// TIA Portal V17 export
// export: Created 2023-05-12T10:40:25.6107869Z, DisplayName Totally Integrated Automation Portal, DisplayVersion V17 Update 4, DisplayName TIA Portal Openness, DisplayVersion V17 Update 4, DisplayName TIA Portal Version Control Interface, DisplayVersion V17, DisplayName STEP 7 Professional, DisplayVersion V17 Update 4, DisplayName STEP 7 Safety, DisplayVersion V17, DisplayName WinCC Advanced / Unified PC, DisplayVersion V17 Update 4
FUNCTION_BLOCK "FB_EM_InputConditioning"   // FB19, LAD
{ S7_Optimized_Access := 'TRUE' }
VERSION : 0.1
// stored: AutoNumber true, CodeModifiedDate 2023-05-12T12:59:41.6492354Z, CompileDate 2023-05-12T12:59:41.6492354Z, CreationDate 2023-05-08T12:19:11.3376827Z, DownloadWithoutReinit false, HandleErrorsWithinBlock false, InterfaceModifiedDate 2023-05-12T12:59:19.7337351Z, IsConsistent true, IsIECCheckEnabled false, IsKnowHowProtected false, IsRetainMemResEnabled false, IsWriteProtected false, LibraryConformanceStatus Warning: The object contains access to global data blocks., MemoryReserve 100, ModifiedDate 2023-05-12T12:59:41.6492354Z, ParameterModified 2022-09-13T10:25:33.4387708Z, PLCSimAdvancedSupport true, SetENOAutomatically false, StructureModified 2023-05-12T12:59:19.7337351Z, UDAEnableTagReadback false
   VAR
      TT01_TempZasil_JKK13_Inst { S7_SetPoint := 'True'} : "FB_CM_MeasurementPoint";
      TT02_TempPowr_JKK13_Inst { S7_SetPoint := 'True'} : "FB_CM_MeasurementPoint";
      TT03_TemZasil_SPC_Kart_Inst { S7_SetPoint := 'True'} : "FB_CM_MeasurementPoint";
      TT04_TempPowr_SPC_Kart_Inst { S7_SetPoint := 'True'} : "FB_CM_MeasurementPoint";
      TT05_TempZasil_SC_Rogacz_Inst { S7_SetPoint := 'True'} : "FB_CM_MeasurementPoint";
      TT06_TempPowr_SC_Rogacz_Inst { S7_SetPoint := 'True'} : "FB_CM_MeasurementPoint";
      PT01_CisnZasil_JKK13_Inst { S7_SetPoint := 'True'} : "FB_CM_MeasurementPoint";
      PT02_CisnPowr_JKK13_Inst { S7_SetPoint := 'True'} : "FB_CM_MeasurementPoint";
      PT03_CisnZasil_SPC_Kart_Inst { S7_SetPoint := 'True'} : "FB_CM_MeasurementPoint";
      PT04_CisnPowr_SPC_Kart_Inst { S7_SetPoint := 'True'} : "FB_CM_MeasurementPoint";
      PT05_CisnZasil_SC_Rogacz_Inst { S7_SetPoint := 'True'} : "FB_CM_MeasurementPoint";
      PT06_CisnPowr_SC_Rogacz_Inst { S7_SetPoint := 'True'} : "FB_CM_MeasurementPoint";
      TTs_TempSzafy_Inst { S7_SetPoint := 'True'} : "FB_CM_MeasurementPoint";
      TTk_TempKom_Inst { S7_SetPoint := 'True'} : "FB_CM_MeasurementPoint";
      TTz_TempZewn_Inst { S7_SetPoint := 'True'} : "FB_CM_MeasurementPoint";
      Rezerwa1_Inst { S7_SetPoint := 'True'} : "FB_CM_MeasurementPoint";
   END_VAR
BEGIN

REGION Network 1: TT01_TempZasil_JKK13 - Temperatura zasilania z JKK13
   // TT01_TempZasil_JKK13 - Temperatura zasilania z JKK13
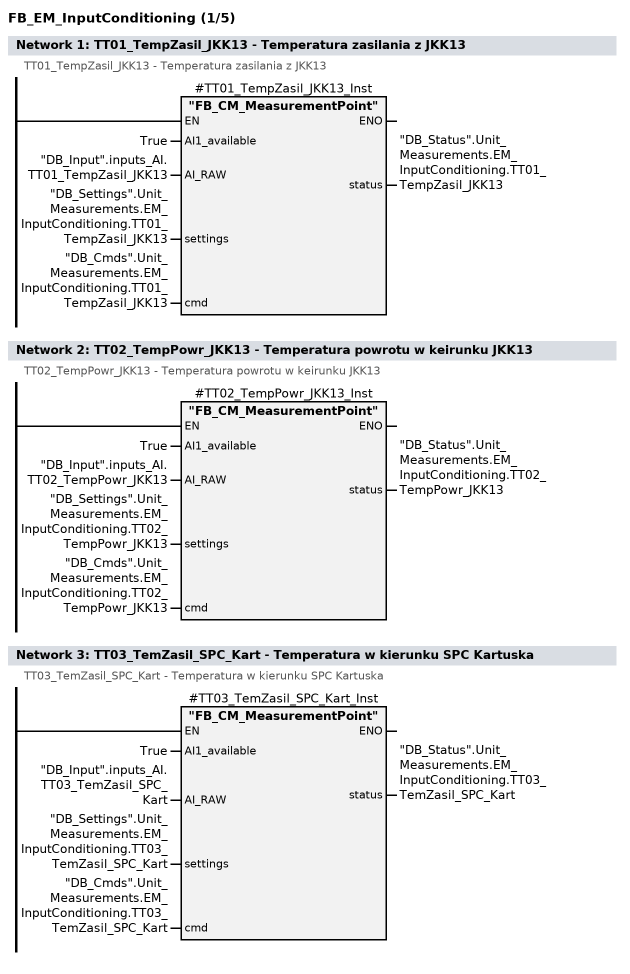
   RUNG wire#powerrail
      #TT01_TempZasil_JKK13_Inst(AI1_available := True, AI_RAW := "DB_Input".inputs_AI.TT01_TempZasil_JKK13, settings := "DB_Settings".Unit_Measurements.EM_InputConditioning.TT01_TempZasil_JKK13, cmd := "DB_Cmds".Unit_Measurements.EM_InputConditioning.TT01_TempZasil_JKK13, status => "DB_Status".Unit_Measurements.EM_InputConditioning.TT01_TempZasil_JKK13)
   END_RUNG
   // the same network as SCL:
   #TT01_TempZasil_JKK13_Inst(AI1_available := True,   // "FB_CM_MeasurementPoint"
                           AI_RAW := "DB_Input".inputs_AI.TT01_TempZasil_JKK13,
                           settings := "DB_Settings".Unit_Measurements.EM_InputConditioning.TT01_TempZasil_JKK13,
                           cmd := "DB_Cmds".Unit_Measurements.EM_InputConditioning.TT01_TempZasil_JKK13,
                           status => "DB_Status".Unit_Measurements.EM_InputConditioning.TT01_TempZasil_JKK13);
END_REGION

REGION Network 2: TT02_TempPowr_JKK13 - Temperatura powrotu w keirunku JKK13
   // TT02_TempPowr_JKK13 - Temperatura powrotu w keirunku JKK13
   RUNG wire#powerrail
      #TT02_TempPowr_JKK13_Inst(AI1_available := True, AI_RAW := "DB_Input".inputs_AI.TT02_TempPowr_JKK13, settings := "DB_Settings".Unit_Measurements.EM_InputConditioning.TT02_TempPowr_JKK13, cmd := "DB_Cmds".Unit_Measurements.EM_InputConditioning.TT02_TempPowr_JKK13, status => "DB_Status".Unit_Measurements.EM_InputConditioning.TT02_TempPowr_JKK13)
   END_RUNG
   // the same network as SCL:
   #TT02_TempPowr_JKK13_Inst(AI1_available := True,   // "FB_CM_MeasurementPoint"
                           AI_RAW := "DB_Input".inputs_AI.TT02_TempPowr_JKK13,
                           settings := "DB_Settings".Unit_Measurements.EM_InputConditioning.TT02_TempPowr_JKK13,
                           cmd := "DB_Cmds".Unit_Measurements.EM_InputConditioning.TT02_TempPowr_JKK13,
                           status => "DB_Status".Unit_Measurements.EM_InputConditioning.TT02_TempPowr_JKK13);
END_REGION

REGION Network 3: TT03_TemZasil_SPC_Kart - Temperatura w kierunku SPC Kartuska
   // TT03_TemZasil_SPC_Kart - Temperatura w kierunku SPC Kartuska
   RUNG wire#powerrail
      #TT03_TemZasil_SPC_Kart_Inst(AI1_available := True, AI_RAW := "DB_Input".inputs_AI.TT03_TemZasil_SPC_Kart, settings := "DB_Settings".Unit_Measurements.EM_InputConditioning.TT03_TemZasil_SPC_Kart, cmd := "DB_Cmds".Unit_Measurements.EM_InputConditioning.TT03_TemZasil_SPC_Kart, status => "DB_Status".Unit_Measurements.EM_InputConditioning.TT03_TemZasil_SPC_Kart)
   END_RUNG
   // the same network as SCL:
   #TT03_TemZasil_SPC_Kart_Inst(AI1_available := True,   // "FB_CM_MeasurementPoint"
                           AI_RAW := "DB_Input".inputs_AI.TT03_TemZasil_SPC_Kart,
                           settings := "DB_Settings".Unit_Measurements.EM_InputConditioning.TT03_TemZasil_SPC_Kart,
                           cmd := "DB_Cmds".Unit_Measurements.EM_InputConditioning.TT03_TemZasil_SPC_Kart,
                           status => "DB_Status".Unit_Measurements.EM_InputConditioning.TT03_TemZasil_SPC_Kart);
END_REGION

REGION Network 4: TT04_TempPowr_SPC_Kart - Temperatura powrotu z SPC Kartuska
   // TT04_TempPowr_SPC_Kart - Temperatura powrotu z SPC Kartuska
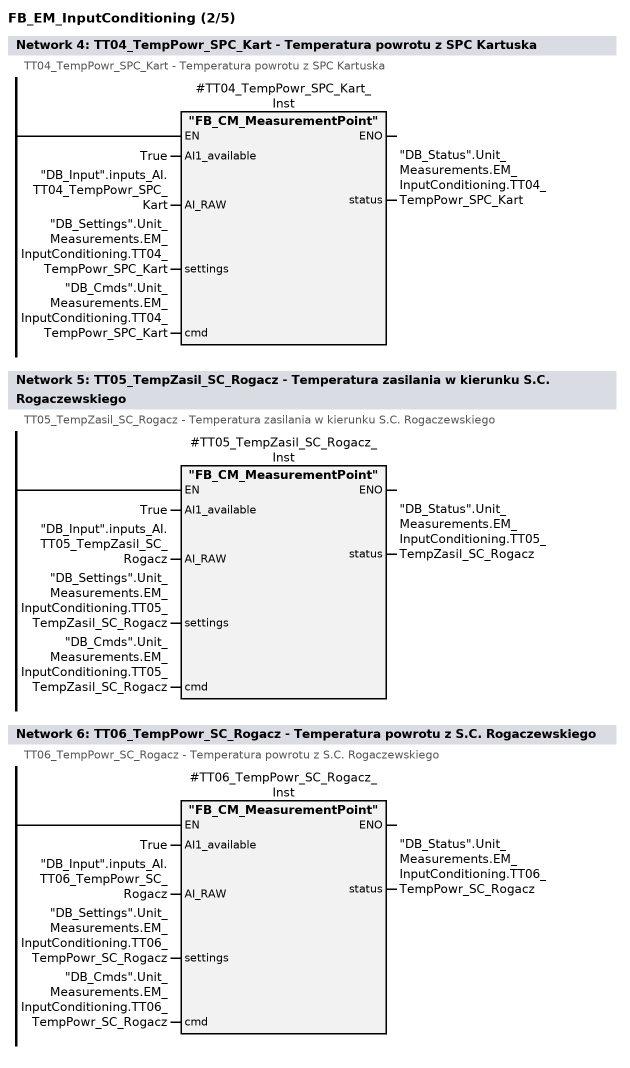
   RUNG wire#powerrail
      #TT04_TempPowr_SPC_Kart_Inst(AI1_available := True, AI_RAW := "DB_Input".inputs_AI.TT04_TempPowr_SPC_Kart, settings := "DB_Settings".Unit_Measurements.EM_InputConditioning.TT04_TempPowr_SPC_Kart, cmd := "DB_Cmds".Unit_Measurements.EM_InputConditioning.TT04_TempPowr_SPC_Kart, status => "DB_Status".Unit_Measurements.EM_InputConditioning.TT04_TempPowr_SPC_Kart)
   END_RUNG
   // the same network as SCL:
   #TT04_TempPowr_SPC_Kart_Inst(AI1_available := True,   // "FB_CM_MeasurementPoint"
                           AI_RAW := "DB_Input".inputs_AI.TT04_TempPowr_SPC_Kart,
                           settings := "DB_Settings".Unit_Measurements.EM_InputConditioning.TT04_TempPowr_SPC_Kart,
                           cmd := "DB_Cmds".Unit_Measurements.EM_InputConditioning.TT04_TempPowr_SPC_Kart,
                           status => "DB_Status".Unit_Measurements.EM_InputConditioning.TT04_TempPowr_SPC_Kart);
END_REGION

REGION Network 5: TT05_TempZasil_SC_Rogacz - Temperatura zasilania w kierunku S.C. Rogaczewskiego
   // TT05_TempZasil_SC_Rogacz - Temperatura zasilania w kierunku S.C. Rogaczewskiego
   RUNG wire#powerrail
      #TT05_TempZasil_SC_Rogacz_Inst(AI1_available := True, AI_RAW := "DB_Input".inputs_AI.TT05_TempZasil_SC_Rogacz, settings := "DB_Settings".Unit_Measurements.EM_InputConditioning.TT05_TempZasil_SC_Rogacz, cmd := "DB_Cmds".Unit_Measurements.EM_InputConditioning.TT05_TempZasil_SC_Rogacz, status => "DB_Status".Unit_Measurements.EM_InputConditioning.TT05_TempZasil_SC_Rogacz)
   END_RUNG
   // the same network as SCL:
   #TT05_TempZasil_SC_Rogacz_Inst(AI1_available := True,   // "FB_CM_MeasurementPoint"
                           AI_RAW := "DB_Input".inputs_AI.TT05_TempZasil_SC_Rogacz,
                           settings := "DB_Settings".Unit_Measurements.EM_InputConditioning.TT05_TempZasil_SC_Rogacz,
                           cmd := "DB_Cmds".Unit_Measurements.EM_InputConditioning.TT05_TempZasil_SC_Rogacz,
                           status => "DB_Status".Unit_Measurements.EM_InputConditioning.TT05_TempZasil_SC_Rogacz);
END_REGION

REGION Network 6: TT06_TempPowr_SC_Rogacz - Temperatura powrotu z S.C. Rogaczewskiego
   // TT06_TempPowr_SC_Rogacz - Temperatura powrotu z S.C. Rogaczewskiego
   RUNG wire#powerrail
      #TT06_TempPowr_SC_Rogacz_Inst(AI1_available := True, AI_RAW := "DB_Input".inputs_AI.TT06_TempPowr_SC_Rogacz, settings := "DB_Settings".Unit_Measurements.EM_InputConditioning.TT06_TempPowr_SC_Rogacz, cmd := "DB_Cmds".Unit_Measurements.EM_InputConditioning.TT06_TempPowr_SC_Rogacz, status => "DB_Status".Unit_Measurements.EM_InputConditioning.TT06_TempPowr_SC_Rogacz)
   END_RUNG
   // the same network as SCL:
   #TT06_TempPowr_SC_Rogacz_Inst(AI1_available := True,   // "FB_CM_MeasurementPoint"
                           AI_RAW := "DB_Input".inputs_AI.TT06_TempPowr_SC_Rogacz,
                           settings := "DB_Settings".Unit_Measurements.EM_InputConditioning.TT06_TempPowr_SC_Rogacz,
                           cmd := "DB_Cmds".Unit_Measurements.EM_InputConditioning.TT06_TempPowr_SC_Rogacz,
                           status => "DB_Status".Unit_Measurements.EM_InputConditioning.TT06_TempPowr_SC_Rogacz);
END_REGION

REGION Network 7: PT01_CisnZasil_JKK13 - CIśnienie zasilania z JKK13
   // PT01_CisnZasil_JKK13 - CIśnienie zasilania z JKK13
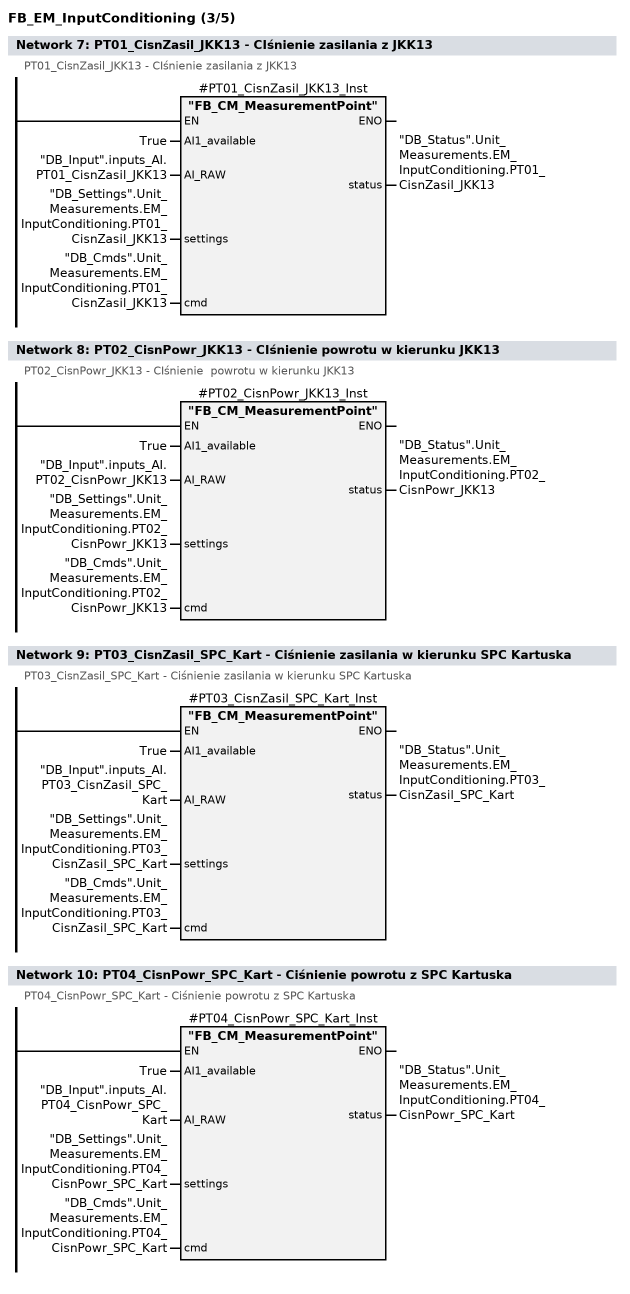
   RUNG wire#powerrail
      #PT01_CisnZasil_JKK13_Inst(AI1_available := True, AI_RAW := "DB_Input".inputs_AI.PT01_CisnZasil_JKK13, settings := "DB_Settings".Unit_Measurements.EM_InputConditioning.PT01_CisnZasil_JKK13, cmd := "DB_Cmds".Unit_Measurements.EM_InputConditioning.PT01_CisnZasil_JKK13, status => "DB_Status".Unit_Measurements.EM_InputConditioning.PT01_CisnZasil_JKK13)
   END_RUNG
   // the same network as SCL:
   #PT01_CisnZasil_JKK13_Inst(AI1_available := True,   // "FB_CM_MeasurementPoint"
                           AI_RAW := "DB_Input".inputs_AI.PT01_CisnZasil_JKK13,
                           settings := "DB_Settings".Unit_Measurements.EM_InputConditioning.PT01_CisnZasil_JKK13,
                           cmd := "DB_Cmds".Unit_Measurements.EM_InputConditioning.PT01_CisnZasil_JKK13,
                           status => "DB_Status".Unit_Measurements.EM_InputConditioning.PT01_CisnZasil_JKK13);
END_REGION

REGION Network 8: PT02_CisnPowr_JKK13 - CIśnienie powrotu w kierunku JKK13
   // PT02_CisnPowr_JKK13 - CIśnienie  powrotu w kierunku JKK13
   RUNG wire#powerrail
      #PT02_CisnPowr_JKK13_Inst(AI1_available := True, AI_RAW := "DB_Input".inputs_AI.PT02_CisnPowr_JKK13, settings := "DB_Settings".Unit_Measurements.EM_InputConditioning.PT02_CisnPowr_JKK13, cmd := "DB_Cmds".Unit_Measurements.EM_InputConditioning.PT02_CisnPowr_JKK13, status => "DB_Status".Unit_Measurements.EM_InputConditioning.PT02_CisnPowr_JKK13)
   END_RUNG
   // the same network as SCL:
   #PT02_CisnPowr_JKK13_Inst(AI1_available := True,   // "FB_CM_MeasurementPoint"
                           AI_RAW := "DB_Input".inputs_AI.PT02_CisnPowr_JKK13,
                           settings := "DB_Settings".Unit_Measurements.EM_InputConditioning.PT02_CisnPowr_JKK13,
                           cmd := "DB_Cmds".Unit_Measurements.EM_InputConditioning.PT02_CisnPowr_JKK13,
                           status => "DB_Status".Unit_Measurements.EM_InputConditioning.PT02_CisnPowr_JKK13);
END_REGION

REGION Network 9: PT03_CisnZasil_SPC_Kart - Ciśnienie zasilania w kierunku SPC Kartuska
   // PT03_CisnZasil_SPC_Kart - Ciśnienie zasilania w kierunku SPC Kartuska
   RUNG wire#powerrail
      #PT03_CisnZasil_SPC_Kart_Inst(AI1_available := True, AI_RAW := "DB_Input".inputs_AI.PT03_CisnZasil_SPC_Kart, settings := "DB_Settings".Unit_Measurements.EM_InputConditioning.PT03_CisnZasil_SPC_Kart, cmd := "DB_Cmds".Unit_Measurements.EM_InputConditioning.PT03_CisnZasil_SPC_Kart, status => "DB_Status".Unit_Measurements.EM_InputConditioning.PT03_CisnZasil_SPC_Kart)
   END_RUNG
   // the same network as SCL:
   #PT03_CisnZasil_SPC_Kart_Inst(AI1_available := True,   // "FB_CM_MeasurementPoint"
                           AI_RAW := "DB_Input".inputs_AI.PT03_CisnZasil_SPC_Kart,
                           settings := "DB_Settings".Unit_Measurements.EM_InputConditioning.PT03_CisnZasil_SPC_Kart,
                           cmd := "DB_Cmds".Unit_Measurements.EM_InputConditioning.PT03_CisnZasil_SPC_Kart,
                           status => "DB_Status".Unit_Measurements.EM_InputConditioning.PT03_CisnZasil_SPC_Kart);
END_REGION

REGION Network 10: PT04_CisnPowr_SPC_Kart - Ciśnienie powrotu z SPC Kartuska
   // PT04_CisnPowr_SPC_Kart - Ciśnienie powrotu z SPC Kartuska
   RUNG wire#powerrail
      #PT04_CisnPowr_SPC_Kart_Inst(AI1_available := True, AI_RAW := "DB_Input".inputs_AI.PT04_CisnPowr_SPC_Kart, settings := "DB_Settings".Unit_Measurements.EM_InputConditioning.PT04_CisnPowr_SPC_Kart, cmd := "DB_Cmds".Unit_Measurements.EM_InputConditioning.PT04_CisnPowr_SPC_Kart, status => "DB_Status".Unit_Measurements.EM_InputConditioning.PT04_CisnPowr_SPC_Kart)
   END_RUNG
   // the same network as SCL:
   #PT04_CisnPowr_SPC_Kart_Inst(AI1_available := True,   // "FB_CM_MeasurementPoint"
                           AI_RAW := "DB_Input".inputs_AI.PT04_CisnPowr_SPC_Kart,
                           settings := "DB_Settings".Unit_Measurements.EM_InputConditioning.PT04_CisnPowr_SPC_Kart,
                           cmd := "DB_Cmds".Unit_Measurements.EM_InputConditioning.PT04_CisnPowr_SPC_Kart,
                           status => "DB_Status".Unit_Measurements.EM_InputConditioning.PT04_CisnPowr_SPC_Kart);
END_REGION

REGION Network 11: PT05_CisnZasil_SC_Rogacz - Ciśnienie zasilania w kierunku S.C Rogaczewskiego
   // PT05_CisnZasil_SC_Rogacz - Ciśnienie zasilania w kierunku S.C Rogaczewskiego
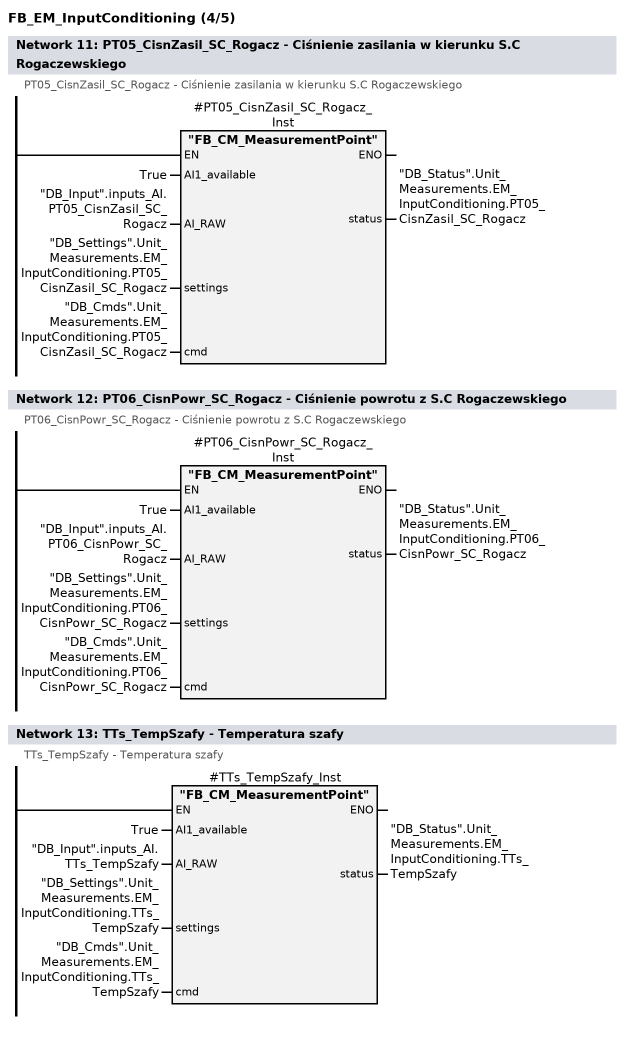
   RUNG wire#powerrail
      #PT05_CisnZasil_SC_Rogacz_Inst(AI1_available := True, AI_RAW := "DB_Input".inputs_AI.PT05_CisnZasil_SC_Rogacz, settings := "DB_Settings".Unit_Measurements.EM_InputConditioning.PT05_CisnZasil_SC_Rogacz, cmd := "DB_Cmds".Unit_Measurements.EM_InputConditioning.PT05_CisnZasil_SC_Rogacz, status => "DB_Status".Unit_Measurements.EM_InputConditioning.PT05_CisnZasil_SC_Rogacz)
   END_RUNG
   // the same network as SCL:
   #PT05_CisnZasil_SC_Rogacz_Inst(AI1_available := True,   // "FB_CM_MeasurementPoint"
                           AI_RAW := "DB_Input".inputs_AI.PT05_CisnZasil_SC_Rogacz,
                           settings := "DB_Settings".Unit_Measurements.EM_InputConditioning.PT05_CisnZasil_SC_Rogacz,
                           cmd := "DB_Cmds".Unit_Measurements.EM_InputConditioning.PT05_CisnZasil_SC_Rogacz,
                           status => "DB_Status".Unit_Measurements.EM_InputConditioning.PT05_CisnZasil_SC_Rogacz);
END_REGION

REGION Network 12: PT06_CisnPowr_SC_Rogacz - Ciśnienie powrotu z S.C Rogaczewskiego
   // PT06_CisnPowr_SC_Rogacz - Ciśnienie powrotu z S.C Rogaczewskiego
   RUNG wire#powerrail
      #PT06_CisnPowr_SC_Rogacz_Inst(AI1_available := True, AI_RAW := "DB_Input".inputs_AI.PT06_CisnPowr_SC_Rogacz, settings := "DB_Settings".Unit_Measurements.EM_InputConditioning.PT06_CisnPowr_SC_Rogacz, cmd := "DB_Cmds".Unit_Measurements.EM_InputConditioning.PT06_CisnPowr_SC_Rogacz, status => "DB_Status".Unit_Measurements.EM_InputConditioning.PT06_CisnPowr_SC_Rogacz)
   END_RUNG
   // the same network as SCL:
   #PT06_CisnPowr_SC_Rogacz_Inst(AI1_available := True,   // "FB_CM_MeasurementPoint"
                           AI_RAW := "DB_Input".inputs_AI.PT06_CisnPowr_SC_Rogacz,
                           settings := "DB_Settings".Unit_Measurements.EM_InputConditioning.PT06_CisnPowr_SC_Rogacz,
                           cmd := "DB_Cmds".Unit_Measurements.EM_InputConditioning.PT06_CisnPowr_SC_Rogacz,
                           status => "DB_Status".Unit_Measurements.EM_InputConditioning.PT06_CisnPowr_SC_Rogacz);
END_REGION

REGION Network 13: TTs_TempSzafy - Temperatura szafy
   // TTs_TempSzafy - Temperatura szafy
   RUNG wire#powerrail
      #TTs_TempSzafy_Inst(AI1_available := True, AI_RAW := "DB_Input".inputs_AI.TTs_TempSzafy, settings := "DB_Settings".Unit_Measurements.EM_InputConditioning.TTs_TempSzafy, cmd := "DB_Cmds".Unit_Measurements.EM_InputConditioning.TTs_TempSzafy, status => "DB_Status".Unit_Measurements.EM_InputConditioning.TTs_TempSzafy)
   END_RUNG
   // the same network as SCL:
   #TTs_TempSzafy_Inst(AI1_available := True,   // "FB_CM_MeasurementPoint"
                       AI_RAW := "DB_Input".inputs_AI.TTs_TempSzafy,
                       settings := "DB_Settings".Unit_Measurements.EM_InputConditioning.TTs_TempSzafy,
                       cmd := "DB_Cmds".Unit_Measurements.EM_InputConditioning.TTs_TempSzafy,
                       status => "DB_Status".Unit_Measurements.EM_InputConditioning.TTs_TempSzafy);
END_REGION

REGION Network 14: TTk_TempKom - Temperatura w komorze
   // TTk_TempKom - Temperatura w komorze
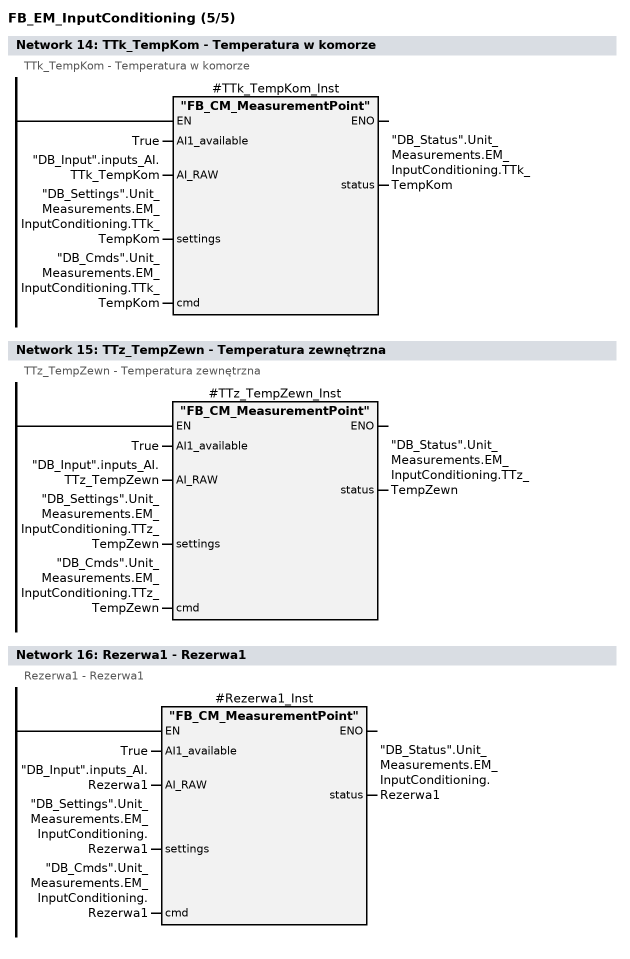
   RUNG wire#powerrail
      #TTk_TempKom_Inst(AI1_available := True, AI_RAW := "DB_Input".inputs_AI.TTk_TempKom, settings := "DB_Settings".Unit_Measurements.EM_InputConditioning.TTk_TempKom, cmd := "DB_Cmds".Unit_Measurements.EM_InputConditioning.TTk_TempKom, status => "DB_Status".Unit_Measurements.EM_InputConditioning.TTk_TempKom)
   END_RUNG
   // the same network as SCL:
   #TTk_TempKom_Inst(AI1_available := True,   // "FB_CM_MeasurementPoint"
                     AI_RAW := "DB_Input".inputs_AI.TTk_TempKom,
                     settings := "DB_Settings".Unit_Measurements.EM_InputConditioning.TTk_TempKom,
                     cmd := "DB_Cmds".Unit_Measurements.EM_InputConditioning.TTk_TempKom,
                     status => "DB_Status".Unit_Measurements.EM_InputConditioning.TTk_TempKom);
END_REGION

REGION Network 15: TTz_TempZewn - Temperatura zewnętrzna
   // TTz_TempZewn - Temperatura zewnętrzna
   RUNG wire#powerrail
      #TTz_TempZewn_Inst(AI1_available := True, AI_RAW := "DB_Input".inputs_AI.TTz_TempZewn, settings := "DB_Settings".Unit_Measurements.EM_InputConditioning.TTz_TempZewn, cmd := "DB_Cmds".Unit_Measurements.EM_InputConditioning.TTz_TempZewn, status => "DB_Status".Unit_Measurements.EM_InputConditioning.TTz_TempZewn)
   END_RUNG
   // the same network as SCL:
   #TTz_TempZewn_Inst(AI1_available := True,   // "FB_CM_MeasurementPoint"
                      AI_RAW := "DB_Input".inputs_AI.TTz_TempZewn,
                      settings := "DB_Settings".Unit_Measurements.EM_InputConditioning.TTz_TempZewn,
                      cmd := "DB_Cmds".Unit_Measurements.EM_InputConditioning.TTz_TempZewn,
                      status => "DB_Status".Unit_Measurements.EM_InputConditioning.TTz_TempZewn);
END_REGION

REGION Network 16: Rezerwa1 - Rezerwa1
   // Rezerwa1 - Rezerwa1
   RUNG wire#powerrail
      #Rezerwa1_Inst(AI1_available := True, AI_RAW := "DB_Input".inputs_AI.Rezerwa1, settings := "DB_Settings".Unit_Measurements.EM_InputConditioning.Rezerwa1, cmd := "DB_Cmds".Unit_Measurements.EM_InputConditioning.Rezerwa1, status => "DB_Status".Unit_Measurements.EM_InputConditioning.Rezerwa1)
   END_RUNG
   // the same network as SCL:
   #Rezerwa1_Inst(AI1_available := True,   // "FB_CM_MeasurementPoint"
                  AI_RAW := "DB_Input".inputs_AI.Rezerwa1,
                  settings := "DB_Settings".Unit_Measurements.EM_InputConditioning.Rezerwa1,
                  cmd := "DB_Cmds".Unit_Measurements.EM_InputConditioning.Rezerwa1,
                  status => "DB_Status".Unit_Measurements.EM_InputConditioning.Rezerwa1);
END_REGION
END_FUNCTION_BLOCK
